//{attribute 'qualified_only'}   //enable this if you want to have qualified global variables, ex: GVL_IO.BoolRelayArray[]
VAR_GLOBAL
	BoolRelayArray  AT %Q* :ARRAY[1..22] OF BOOL;
	//BoolRelayArray AT %QX0.0 :ARRAY[1..21] OF BOOL;
END_VAR

(* stored: Version 1.1.0.1, ProductVersion 3.1.4024.13
   GVL GVL_IO: Id {7d284c7f-20a0-4e3e-8fbe-e0adf73714e3} *)
